TYPE ST_STATION_LIST_RESULT :
STRUCT
  wState    : WORD;   // wState == 0 --> all ok
  nIndex    : ULINT;
  stData    : ST_STATION_MOVER_DATA;  // copy of list entry
END_STRUCT
END_TYPE

(* stored: Version 1.1.0.1, ProductVersion 3.1.4026.13
   DUT ST_STATION_LIST_RESULT: Id {c264fd93-3d8b-446d-b835-f3bfb9bfb8e1} *)
